(* CoDeSys 2.3 export: SENSOR_FOTO.EXP *)

(* Data type *)
TYPE Sensor_Foto :
STRUCT
	Activo : BOOL;
END_STRUCT
END_TYPE
